TYPE ST_PNController_Events :
STRUCT
	b_HeartBeatLost				:	BOOL;
	b_DataConfigurationFault	:	BOOL;
	b_NetworkConfigurationFault	:	BOOL;
	b_DeviceFault				:	BOOL;
END_STRUCT
END_TYPE

(* stored: Version 1.1.0.1, ProductVersion 3.1.4024.12
   DUT ST_PNController_Events: Id {fab317f0-218d-47b3-85fc-35836b4482d1} *)
